// TwinCAT 3 PLC project Untitled1
// ProgramVersion: 3.1.4024.0
// libraries:
//   Tc2_Standard, * (Beckhoff Automation GmbH)
//   Tc2_System, * (Beckhoff Automation GmbH)
//   Tc2_Utilities, * (Beckhoff Automation GmbH)
//   Tc3_Module, * (Beckhoff Automation GmbH)
// project tree:
//   DUTs/ ST_ProfinetDiagnostics.TcDUT, ST_SerialDevice_Alarms.TcDUT, ST_VantagePro_Alarms.TcDUT, U_ByteToString.TcDUT, U_ReceivedData.TcDUT
//   GVLs/ GVL_Test.TcGVL
//   / PlcTask.TcTTO
//   POUs/ FB_TestMethods.TcPOU, F_RealIsValid.TcPOU, F_RealIsNaN.TcPOU, F_REAL_TO_STRING.TcPOU, F_Round_REAL.TcPOU, MAIN.TcPOU, Test_1.TcPOU, Test_2.TcPOU
// real-time tasks:
//   TASK PlcTask: cycle T#8ms, priority 20, ADS port 350
// I/O:
//   DEVICE Device 2 (EtherCAT) (disabled), AmsNetId 192.168.188.130.3.1
//     Term 3 (EK1200) [EK1200-5000 EtherCAT Power supply (2A E-Bus)]
//       Term 4 (EL6900) [EL6900, TwinSAFE PLC]
//   DEVICE Device 1 (EtherCAT Automation Protocol) (disabled), AmsNetId 192.168.188.130.2.1
//     FromConveyor (Subscriber)
//     ToConveyor (Publisher)
// variable links:
//   Device 1 (EtherCAT Automation Protocol) <-> Device 2 (EtherCAT)/Term 3 (EK1200)/Term 4 (EL6900)
//     ToConveyor (Publisher)/PubFSoE/Outputs/VarData <-> ConnectionInputs/Message_2 TxPDO
//   Device 2 (EtherCAT) <-> Device 1 (EtherCAT Automation Protocol)/FromConveyor (Subscriber)
//     Term 3 (EK1200)/Term 4 (EL6900)/ConnectionOutputs/Message_2 RxPDO <-> SubFSoE/Inputs/VarData
//   Untitled1/Untitled1 Instance <-> Device 2 (EtherCAT)/Term 3 (EK1200)/Term 4 (EL6900)
//     PlcTask Inputs/MAIN.FSoE{1..4} <-> StandardInputs/Standard Out Var {3..6}  (4 links)
//     PlcTask Outputs/MAIN.err_ack <-> StandardOutputs/Standard In Var 1

CONFIGURATION Untitled1
    RESOURCE PLC ON TwinCAT3
        TASK PlcTask(INTERVAL := T#10ms, PRIORITY := 20);
        PROGRAM MAIN WITH PlcTask : MAIN;
    END_RESOURCE
END_CONFIGURATION

// ---- DUTs/ST_ProfinetDiagnostics.TcDUT
TYPE ST_ProfinetDiagnostics :
STRUCT
	PnIoBoxState			AT %I* : UINT;
	PnIoBoxDiag				AT %I* : UINT;
	PnIoBoxCtrl				AT %Q* : UINT;
END_STRUCT
END_TYPE

// ---- DUTs/ST_SerialDevice_Alarms.TcDUT
TYPE ST_SerialDevice_Alarms :
STRUCT
	bAdsError			: BOOL;
	nAdsErrorID		    : UDINT;
	bComPortNotOpen	    : BOOL;
	nReceiveError		: INT;
	bReceiveTimeout	    : BOOL;
	bSendError		    : BOOL;
	nSendErrorID		: INT;
	bCommsNotOK		    : BOOL;
	nRxError			: UDINT;
	nTxError			: UDINT;

END_STRUCT
END_TYPE

// ---- DUTs/ST_VantagePro_Alarms.TcDUT
TYPE ST_VantagePro_Alarms EXTENDS ST_SerialDevice_Alarms:
STRUCT
END_STRUCT
END_TYPE

// ---- DUTs/U_ByteToString.TcDUT
TYPE U_ByteToString :
UNION
	byteArrayValue		: ARRAY[0..99] OF BYTE;
	stringValue			: STRING(99);
	realValue			: REAL;
	wordValue			: WORD;
END_UNION
END_TYPE

// ---- DUTs/U_ReceivedData.TcDUT
TYPE U_ReceivedData :
UNION
	DataArray	: ARRAY[0 .. 255] OF BYTE;
	DataString	: STRING(255);
END_UNION
END_TYPE

// ---- GVLs/GVL_Test.TcGVL
{attribute 'qualified_only'}
VAR_GLOBAL
	Bool1		: BOOL;
	Bool2		: BOOL;
	Bool3		: BOOL;
	
	Word1		: WORD;
	Word2		: WORD;
	Word3		: WORD;
	
	Real1		: REAL;
	Real2		: REAL;
	Real3		: REAL;
	
	Dint1		: DINT;
	Dint2		: DINT;
	Dint3		: DINT;
	
	arrByte		: ARRAY[1..100] OF BYTE;
	
	alarmGVL		: ST_VantagePro_Alarms; (* := (bAdsError := FALSE, nAdsErrorID := 0,
													bComPortNotOpen := FALSE, nReceiveError := 0,
													bReceiveTimeout := FALSE, bSendError := FALSE,
													nSendErrorID := 0, bCommsNotOK := FALSE,
													nRxError := 0, nTxError := 0);*)
END_VAR

// ---- POUs/MAIN.TcPOU
PROGRAM MAIN
VAR
	rInternalDistanceMastering	: REAL;
	iDataByte1		: BYTE;
	iDataByte2		: BYTE;
	iDataByte3		: BYTE;
	dwordtest		: DWORD := 90000;
	uString		: U_ReceivedData;	

	err_ack		AT %Q* : BOOL;
	FSoE1		AT %I* : BOOL;	
	FSoE2		AT %I* : BOOL;	
	FSoE3		AT %I* : BOOL;	
	FSoE4		AT %I* : BOOL;	
	FSoEout		AT %Q* : BOOL;	

	io				: ST_ProfinetDiagnostics;	

	refTest1		: Test_1;
	refTest2		: Test_1;	
	refTest3		: Test_2;	
	
	Iotest			AT %I* : BOOL;

	rWindSpeed		: REAL;
	rWindDirection	: REAL;
	iStatusCode		: INT;
	sResult			: STRING;
	uniontest		: U_ByteToString;	

	iNanWord1		: WORD;
	iNanWord2		: WORD;
	aNaNarray		: ARRAY[1..32] OF BOOL;
	iNanDint		: DINT;
	rNanTest		: REAL;
	bNanResult		: BOOL;
	refReal			: REFERENCE TO REAL;
	
	

	arr				: ARRAY[1..10] OF BYTE;	
	arrTest			: BOOL;
	arrRead			: BOOL;

	rReal			: REAL;
	rRoundedReal	: REAL;
	prec			: INT;
	stringTest1		: STRING;
	stringTest2		: STRING;
	
	iPrecision		: INT;
	iTempInt		: DINT;
	iWholeNum		: DINT;
	iDecimal		: DINT;
	
	iAddZeros		: INT;
	
	sOut			: STRING;
	
	i				: INT;


	test 	: ARRAY[0..2] OF BOOL;
	test1	: BOOL;
	testMeth1 : FB_TestMethods;
	testMeth2 : FB_TestMethods;
	testMeth : FB_TestMethods;
	test2000 : BOOL;
	what : INT;
	
	exec	: BOOL;
	
	Run			AT %Q* : BOOL;
	Reset		AT %Q* : BOOL;
	ErrAck		AT %Q* : BOOL;
	
	TestSafeInput2	AT %Q* : BOOL;
	
	t1 : DINT;
	t2 : DINT;
	t3 : DINT;
	t4 : DINT;
	t5 : DINT;
	t6 : DINT;
	
	alarm		: ST_VantagePro_Alarms;
	
	fbWritePersistentData	: FB_WritePersistentData;
	tonWritePersistentData	: TON;
	
	toggle1					: BOOL;
	
	randomBARIABLE		: REAL;
	testMeth3 : FB_TestMethods;
	testMeth4 : FB_TestMethods;
	
    nTaskIdx     : DINT;
    nCycleTime   : UDINT;
	
	limits		: INT(-3..3);
END_VAR
VAR CONSTANT
	alarmCons	: ST_VantagePro_Alarms := ();
END_VAR
VAR_TEMP
	alarmTemp	: ST_VantagePro_Alarms;
END_VAR

iPrecision := BIT_TO_INT(dwordtest.1) * 3;

//iPrecision := 10;
//rInternalDistanceMastering	:= (DWORD_TO_REAL(dwordtest) * 102/65520 - 51)/100 * iPrecision;

//iStatusCode	:= LEN(uString.DataString);

//dwordtest	:= SHL(iDataByte3 AND 2#0011_1111, 12) OR SHL(iDataByte2 AND 2#0011_1111, 6) OR iDataByte1 AND 2#0011_1111;

(*
refTest1();
refTest2();
refTest3();

refTest1.P_IO.PnIoBoxState := io.PnIoBoxState;
refTest1.P_IO.PnIoBoxDiag := io.PnIoBoxDiag;
io.PnIoBoxCtrl := refTest1.P_IO.PnIoBoxCtrl;

refTest1.P_REAL := rWindSpeed;

//refTest2.P_REAL := refTest1.P_REAL;
//refTest3.P_REAL REF= refTest1.P_REAL;

	sResult			:= uniontest.stringValue;
	sResult			:= DELETE(sResult, FIND(sResult, ' '), 1);
	
	rWindSpeed		:= STRING_TO_REAL(LEFT(sResult, FIND(sResult, ' ') - 1));
	sResult			:= DELETE(sResult, FIND(sResult, ' '), 1);
	
	rWindDirection	:= STRING_TO_REAL(LEFT(sResult, FIND(sResult, ' ') - 1));
	sResult			:= DELETE(sResult, FIND(sResult, ' '), 1);
	IF rWindDirection >= 360 THEN
		rWindDirection	:= rWindDirection - 360;
	END_IF
	
	iStatusCode		:= STRING_TO_INT(LEFT(sResult, FIND(sResult, '*') - 1));

iNanDint. 0	:= aNaNarray[ 1];
iNanDint. 1	:= aNaNarray[ 2];
iNanDint. 2	:= aNaNarray[ 3];
iNanDint. 3	:= aNaNarray[ 4];
iNanDint. 4	:= aNaNarray[ 5];
iNanDint. 5	:= aNaNarray[ 6];
iNanDint. 6	:= aNaNarray[ 7];
iNanDint. 7	:= aNaNarray[ 8];
iNanDint. 8	:= aNaNarray[ 9];
iNanDint. 9	:= aNaNarray[10];
iNanDint.10	:= aNaNarray[11];
iNanDint.11	:= aNaNarray[12];
iNanDint.12	:= aNaNarray[13];
iNanDint.13	:= aNaNarray[14];
iNanDint.14	:= aNaNarray[15];
iNanDint.15	:= aNaNarray[16];
iNanDint.16	:= aNaNarray[17];
iNanDint.17	:= aNaNarray[18];
iNanDint.18	:= aNaNarray[19];
iNanDint.19	:= aNaNarray[20];
iNanDint.20	:= aNaNarray[21];
iNanDint.21	:= aNaNarray[22];
iNanDint.22	:= aNaNarray[23];

iNanDint.23	:= aNaNarray[24];
iNanDint.24	:= aNaNarray[25];
iNanDint.25	:= aNaNarray[26];
iNanDint.26	:= aNaNarray[27];
iNanDint.27	:= aNaNarray[28];
iNanDint.28	:= aNaNarray[29];
iNanDint.29	:= aNaNarray[30];
iNanDint.30	:= aNaNarray[31];

iNanDint.31	:= aNaNarray[32];

IF toggle1 THEN
	MEMCPY(ADR(rNanTest), ADR(iNanDint), SIZEOF(iNanDint));
END_IF
	
refReal		REF= rNanTest;

bNanResult	:= F_RealIsNaN(rNanTest);

//bNanResult	:= F_RealIsValid(rInput	:= rNanTest);

//bNanResult	:= RealIsNan(refReal);

//testMeth1(refReal	:= rNanTest);


MEMCPY(ADR(arr), ADR(arrTest), SIZEOF(arrTest));

MEMCPY(ADR(arrRead), ADR(arr[5]), SIZEOF(arrRead));

arr[10]	:= BOOL_TO_BYTE(arrTest);

rRoundedReal	:= F_Round_REAL(rReal,prec);
stringTest1		:= REAL_TO_STRING(rRoundedReal);

stringTest2		:= F_REAL_TO_STRING(rReal,prec);

iPrecision	:= prec;
iTempInt := REAL_TO_DINT(rReal * EXPT(10,ABS(iPrecision)));

iWholeNum	:= TRUNC(iTempInt / EXPT(10,ABS(iPrecision)));

iDecimal	:= iTempInt - LREAL_TO_DINT(iWholeNum * EXPT(10,ABS(iPrecision)));

sOut		:= CONCAT(DINT_TO_STRING(iWholeNum), '.');

IF iDecimal > 0 THEN
	iAddZeros	:= ABS(iPrecision) - DINT_TO_INT(TRUNC(LOG(iDecimal))) - 1;

	FOR i := 1 TO iAddZeros DO
		sOut	:= CONCAT(sOut,'0');
	END_FOR
	
	sOut	:= CONCAT(sOut, DINT_TO_STRING(iDecimal));
ELSE
	iAddZeros	:= ABS(iPrecision);

	FOR i := 1 TO iAddZeros DO
		sOut	:= CONCAT(sOut,'0');
	END_FOR
END_IF

nTaskIdx := GETCURTASKINDEXEX();
IF nTaskIdx > 0 THEN
    nCycleTime := _TaskInfo[nTaskIdx].CycleTime;
END_IF

test[0] := TRUE;
test[1] := FALSE;
test[2] := TRUE;


(*IF test = TRUE THEN
	test1 := TRUE;
ELSE
	test1 := FALSE;
END_IF*)

testMeth();

IF test2000 THEN
	what := testMeth.METH(Execute	:= exec);
	//test2000 := true;
END_IF

t1 := MEMCMP(ADR(GVL_test.alarmGVL), ADR(alarm), SIZEOF(GVL_test.alarmGVL));
t2 := MEMCMP(ADR(GVL_test.alarmGVL), ADR(alarmCons), SIZEOF(GVL_test.alarmGVL));
t3 := MEMCMP(ADR(GVL_test.alarmGVL), ADR(alarmTemp), SIZEOF(GVL_test.alarmGVL));
t4 := MEMCMP(ADR(alarm), ADR(alarmCons), SIZEOF(alarm));
t5 := MEMCMP(ADR(alarm), ADR(alarmTemp), SIZEOF(alarm));
t6 := MEMCMP(ADR(alarmCons), ADR(alarmTemp), SIZEOF(alarmCons));

////Save persistent data
//tonWritePersistentData(IN := NOT tonWritePersistentData.Q, PT := T#10M);

//fbWritePersistentData(
//    Port         := 851,
//    Start        := tonWritePersistentData.Q OR toggle1,
//    Mode         := SPDM_VAR_BOOST);
*)

END_PROGRAM

// ---- POUs/Test_1.TcPOU
FUNCTION_BLOCK Test_1
VAR_INPUT
END_VAR
VAR_OUTPUT
END_VAR
VAR
	heyo : REAL;
	random: BOOL;
	io				: ST_ProfinetDiagnostics;
	
END_VAR

random := not random;

PROPERTY P_IO : REFERENCE TO ST_ProfinetDiagnostics
GET
P_IO REF= io;
END_GET
END_PROPERTY

PROPERTY PUBLIC P_REAL : REFERENCE TO REAL
GET
P_REAL REF= heyo;
END_GET
END_PROPERTY

END_FUNCTION_BLOCK

// ---- POUs/Test_2.TcPOU
FUNCTION_BLOCK Test_2
VAR_INPUT
END_VAR
VAR_OUTPUT
END_VAR
VAR
	heyo : REFERENCE TO REAL;
	random: BOOL;
	
END_VAR

random := not random;

PROPERTY PUBLIC P_REAL : REFERENCE TO REAL
SET // PUBLIC
heyo REF= P_REAL;
END_SET
END_PROPERTY

END_FUNCTION_BLOCK

// ---- POUs/FB_TestMethods.TcPOU
FUNCTION_BLOCK FB_TestMethods
VAR_INPUT
	refReal		: REFERENCE TO REAL;
END_VAR
VAR_OUTPUT
END_VAR
VAR
	state1			: INT;
	outP	: BOOL;
	
	check	: BOOl;
END_VAR
VAR PERSISTENT
	persistentTest1	: REAL;
	persistentTest2	: INT;
	persistentTest3	: REAL;
END_VAR

//outP	:= RealIsNan(refReal);

CASE state1 OF
	0: 
		;
		
	1:	
		METH(Execute	:= FALSE);
		
		METH(Execute	:= FALSE, done => check);
	
	2:
		//check	:= METH.done;
END_CASE

METHOD METH : int
VAR_INPUT
	Execute	: BOOL;
END_VAR
VAR_OUTPUT
	done	: BOOL;
END_VAR
VAR
	i : DINT;
	Timer	: ton;
END_VAR
VAR_INST
	ExecuteTrig	: R_TRIG;
	
END_VAR
FOR i := 1 TO 100000 BY 1 DO
	Timer(In := TRUE,PT := T#5S);
	IF i = 99999 THEN
		METH := 5;
	END_IF
END_FOR

ExecuteTrig(CLK := Execute);

//outP	:= ExecuteTrig.Q;

done	:= outP;
END_METHOD

END_FUNCTION_BLOCK

// ---- POUs/F_RealIsValid.TcPOU
FUNCTION F_RealIsValid : BOOL
VAR_INPUT
	rInput			: REAL;
END_VAR
VAR
	refReal			: REFERENCE TO REAL;
END_VAR

refReal		REF= rInput;

IF RealIsNan(refReal) THEN
	F_RealIsValid	:= FALSE;
	RETURN;
ELSE
	IF (ABS(refReal) < EXP(-10) AND refReal <> 0) OR ABS(refReal) > EXP(10) THEN
		F_RealIsValid	:= FALSE;
		RETURN;
	ELSE
		F_RealIsValid	:= TRUE;
		RETURN;
	END_IF
END_IF

END_FUNCTION

// ---- POUs/F_RealIsNaN.TcPOU
FUNCTION F_RealIsNaN : BOOL
VAR_INPUT
	rInput			: REAL;
END_VAR
VAR
	iBitWord		: DWORD;
	
	iExponent		: DWORD;
	iExponentMask	: DWORD := 2#0111_1111__1000_0000__0000_0000__0000_0000;
	
	iMantissa		: DWORD := 2#0000_0000__0111_1111__1111_1111__1111_1111;
	iMantissaMask	: DWORD := 2#0000_0000__0111_1111__1111_1111__1111_1111;
END_VAR

MEMCPY(ADR(iBitWord), ADR(rInput), SIZEOF(iBitWord));

iExponent	:= iBitWord AND iExponentMask;

iMantissa	:= iBitWord AND iMantissaMask;

IF iExponent = iExponentMask AND iMantissa <> 0 THEN
	F_RealIsNaN	:= TRUE;
ELSE
	F_RealIsNaN	:= FALSE;
END_IF

END_FUNCTION

// ---- POUs/F_REAL_TO_STRING.TcPOU
FUNCTION F_REAL_TO_STRING : STRING
VAR_INPUT
	rReal			: REAL;
	iPrecision		: INT;
END_VAR
VAR
	iTempInt		: DINT;
	iWholeNum		: DINT;
	iDecimal		: DINT;
	
	iAddZeros		: INT;
	
	sOut			: STRING;
	
	i				: INT;
END_VAR

IF RealIsNaN(rReal) THEN
	RETURN;
END_IF

iTempInt := REAL_TO_DINT(rReal * EXPT(10,ABS(iPrecision)));

iWholeNum	:= TRUNC(iTempInt / EXPT(10,ABS(iPrecision)));

iDecimal	:= iTempInt - LREAL_TO_DINT(iWholeNum * EXPT(10,ABS(iPrecision)));

sOut		:= CONCAT(DINT_TO_STRING(iWholeNum), '.');

IF iDecimal > 0 THEN
	iAddZeros	:= ABS(iPrecision) - DINT_TO_INT(TRUNC(LOG(iDecimal))) - 1;

	FOR i := 1 TO iAddZeros DO
		sOut	:= CONCAT(sOut,'0');
	END_FOR
	
	sOut	:= CONCAT(sOut, DINT_TO_STRING(iDecimal));
ELSE
	iAddZeros	:= ABS(iPrecision);

	FOR i := 1 TO iAddZeros DO
		sOut	:= CONCAT(sOut,'0');
	END_FOR
END_IF

F_REAL_TO_STRING	:= sOut;

END_FUNCTION

// ---- POUs/F_Round_REAL.TcPOU
FUNCTION F_Round_REAL : REAL
VAR_INPUT
	rInReal			: REAL;
	iPrecision		: INT;
END_VAR
VAR
	rOutReal		: REAL;
	rRoundingVal	: REAL; //last digit for rounding purposes
END_VAR

IF RealIsNaN(rInReal) THEN
	RETURN;
END_IF

rOutReal := rInReal * EXPT(10,ABS(iPrecision));

rRoundingVal := rOutReal - DINT_TO_REAL(TRUNC(rOutReal));
IF rRoundingVal >= 0.5 THEN
	rOutReal	:= DINT_TO_REAL(TRUNC(rOutReal)) + 1;
ELSIF rRoundingVal <= -0.5 THEN
	rOutReal	:= DINT_TO_REAL(TRUNC(rOutReal)) - 1;
ELSE
	rOutReal	:= DINT_TO_REAL(TRUNC(rOutReal));
END_IF

F_Round_REAL	:= rOutReal / EXPT(10,ABS(iPrecision));

END_FUNCTION
